FUNCTION_BLOCK _UDINT_TestSuite EXTENDS TcUnit.FB_TestSuite
VAR
END_VAR

TestAddress();
TestClearReference();
TestClone();
TestTypeNameReturnsExpected();
TestIsFloat();
TestIsSigned();
TestMakeReferenceToFollowsReference();
TestMakeReferenceToUpdatesReference();
TestSize();
TestValueReturnsExpectedAfterInit();
TestValueReturnsExpectedAfterChange();
TestSerializeTypeWith();
TestSerializeWith();
TestTryDeserializeFrom();
TestTryMakeReferenceToFollowsReference();
TestTryMakeReferenceToUpdatesReference();

METHOD PUBLIC TestAddress
VAR
    _type : _UDINT(0);
    notExpected : PVOID := 0;
    actual : PVOID;
END_VAR
TEST('TestAddress');

actual := _type.Address;

AssertFalse(
    Condition := (notExpected = actual),
    Message := 'Type did not return a valid address.'
);

TEST_FINISHED();
END_METHOD

METHOD PUBLIC TestClearReference
VAR
    _type : _UDINT(0);
	target : UDINT := 0;
    expected : UDINT := 0;
    actual : UDINT;
END_VAR
TEST('TestClearReference');

_type.MakeReferenceTo(target);
_type.ClearReference();
target := 123;

actual := _type.Value;

AssertEquals(
    Expected := expected,
    Actual := actual,
    Message := 'Value incorrectly followed target change'
);

TEST_FINISHED();
END_METHOD

METHOD PUBLIC TestClone
VAR
    _type : _UDINT(123);
	clone : I_Datatype;
	isValidClone : BOOL;
	compareResult : DINT;
END_VAR
TEST('TestClone');

clone := _type.Clone();

isValidClone := clone <> 0;

IF isValidClone THEN
	compareResult := memcmp(_type.Address, clone.Address, clone.Size);
END_IF

AssertTrue(
	Condition := isValidClone,
	Message := 'Clone did not produce a clone'
);

AssertEquals_DINT(
	Expected := 0,
    Actual := compareResult,
    Message := 'Clone did not return a valid clone.'
);

clone.Dispose();

TEST_FINISHED();
END_METHOD

METHOD PUBLIC TestIsFloat
VAR
    _type : _UDINT(0);
END_VAR
TEST('TestIsFloat');

AssertFalse(
	Condition := _type.IsFloat,
    Message := 'Type did not correctly identify itself as being unsigned'
);

TEST_FINISHED();
END_METHOD

METHOD PUBLIC TestIsSigned
VAR
    _type : _UDINT(0);
END_VAR
TEST('TestIsSigned');

AssertFalse(
	Condition := _type.IsSigned,
    Message := 'Type did not correctly identify itself as being unsigned'
);

TEST_FINISHED();
END_METHOD

METHOD PUBLIC TestMakeReferenceToFollowsReference
VAR
    _type : _UDINT(0);
	target : UDINT := 0;
    expected : UDINT := 123;
    actual : UDINT;
END_VAR
TEST('TestMakeReferenceToFollowsReference');

_type.MakeReferenceTo(target);
target := 123;

actual := _type.Value;

AssertEquals(
    Expected := expected,
    Actual := actual,
    Message := 'Value did not follow target change'
);

TEST_FINISHED();
END_METHOD

METHOD PUBLIC TestMakeReferenceToUpdatesReference
VAR
    _type : _UDINT(0);
	target : UDINT := 0;
    expected : UDINT := 123;
    actual : UDINT;
END_VAR
TEST('TestMakeReferenceToUpdatesReference');

_type.MakeReferenceTo(target);
_type.Value := 123;

actual := target;

AssertEquals(
    Expected := expected,
    Actual := actual,
    Message := 'Value did not update target'
);

TEST_FINISHED();
END_METHOD

METHOD PUBLIC TestSerializeTypeWith
VAR
    _type : _UDINT(0);
    serializer : JsonSerializer;
    expected : STRING(500) := '{"typeName":"UDINT","minValue":0,"maxValue":4294967295,"isSigned":false,"isFloat":false}';
    actual : STRING(500);
END_VAR
TEST('TestSerializeTypeWith');

serializer.Reset();
_type.SerializeTypeWith(serializer);
serializer.TryGetSerializedData(ADR(actual), SIZEOF(actual));

AssertEquals_STRING(
    Expected := expected,
    Actual := actual,
    Message := 'Serialization of type did not return correct string.'
);

TEST_FINISHED();
END_METHOD

METHOD PUBLIC TestSerializeWith
VAR
    _type : _UDINT(123);
    serializer : JsonSerializer;
    expected : STRING := '123';
    actual : STRING(500);
END_VAR
TEST('TestSerializeWith');

serializer.Reset();
_type.SerializeWith(serializer);
serializer.TryGetSerializedData(ADR(actual), SIZEOF(actual));

AssertEquals_STRING(
    Expected := expected,
    Actual := actual,
    Message := 'Serialization of type data did not return correct string.'
);

TEST_FINISHED();
END_METHOD

METHOD PUBLIC TestSize
VAR
    _type : _UDINT(0);
    expected : UDINT := SIZEOF(UDINT);
    actual : UDINT;
END_VAR
TEST('TestSize');

actual := _type.Size;

AssertEquals_UDINT(
    Expected := Expected,
    Actual := actual,
    Message := 'Type did not return the correct size.'
);

TEST_FINISHED();
END_METHOD

METHOD PUBLIC TestTryDeserializeFrom
VAR
    deserializer : JsonDeserializer;
    feedback : DeserializerFeedback;
    json : STRING := '123';
    _type : _UDINT(0);
    expected : UDINT := 123;
    actual : UDINT;
 END_VAR
TEST('TestTryDeserializeFrom');

deserializer.Reset();
deserializer.TryLoad(json);
_type.TryDeserializeFrom(Deserializer, Feedback);

actual := _type.Value;

AssertEquals(
    Expected := expected,
    Actual := actual,
    Message := 'Type did not deserialize correctly.'
);

TEST_FINISHED();
END_METHOD

METHOD PUBLIC TestTryMakeReferenceToFollowsReference
VAR
    _type : _UDINT(0);
	target : _UDINT(0);
    expected : UDINT := 123;
    actual : UDINT;
END_VAR
TEST('TestTryMakeReferenceToFollowsReference');

_type.TryMakeReferenceTo(target);
target.Value := 123;

actual := _type.Value;

AssertEquals(
    Expected := expected,
    Actual := actual,
    Message := 'Value did not follow target change'
);

TEST_FINISHED();
END_METHOD

METHOD PUBLIC TestTryMakeReferenceToUpdatesReference
VAR
    _type : _UDINT(0);
	target : _UDINT(0);
    expected : UDINT := 123;
    actual : UDINT;
END_VAR
TEST('TestTryMakeReferenceToUpdatesReference');

_type.TryMakeReferenceTo(target);
_type.Value := 123;

actual := target.Value;

AssertEquals(
    Expected := expected,
    Actual := actual,
    Message := 'Value did not update target'
);

TEST_FINISHED();
END_METHOD

METHOD PUBLIC TestTypeNameReturnsExpected
VAR
    _type : _UDINT(0);
    expected : STRING := 'UDINT';
    actual : STRING;
END_VAR
TEST('TestTypeNameReturnsExpected');

actual := _type.TypeName;

AssertEquals_STRING(
    Expected := expected,
    Actual := actual,
    Message := 'Type did not return correct iec type.'
);

TEST_FINISHED();
END_METHOD

METHOD PUBLIC TestValueReturnsExpectedAfterChange
VAR
    _type : _UDINT(0);
    expected : UDINT := 123;
    actual : UDINT;
END_VAR
TEST('TestValueReturnsExpectedAfterChange');

_type.Value := 123;

actual := _type.Value;

AssertEquals(
    Expected := expected,
    Actual := actual,
    Message := 'Expected value not returned after change.'
);

TEST_FINISHED();
END_METHOD

METHOD PUBLIC TestValueReturnsExpectedAfterInit
VAR
    _type : _UDINT(123);
    expected : UDINT := 123;
    actual : UDINT;
END_VAR
TEST('TestValueReturnsExpectedAfterInit');

actual := _type.Value;

AssertEquals(
    Expected := expected,
    Actual := actual,
    Message := 'Expected value not returned after Init.'
);

TEST_FINISHED();
END_METHOD

END_FUNCTION_BLOCK

(* stored: Version 1.1.0.1, ProductVersion 3.1.4024.12
   POU _UDINT_TestSuite: Id {2800a6ae-27d3-03ba-3911-8603c59c029a}, SpecialFunc None
   Method TestAddress: Id {99a2019e-ed45-0102-2932-822e518121fe}
   Method TestClearReference: Id {38937dd6-21b3-0552-20da-5c3d3787943e}
   Method TestClone: Id {b4d84e3b-1860-0841-3c59-7c02cd3bd047}
   Method TestIsFloat: Id {6e2992b0-27c6-462d-9092-3abdf0b287bb}
   Method TestIsSigned: Id {a661132e-a505-0f18-0177-1db667ec6b01}
   Method TestMakeReferenceToFollowsReference: Id {47c3d9a3-4886-0583-38d8-1ff279e5076a}
   Method TestMakeReferenceToUpdatesReference: Id {b107d813-75e4-0da0-3145-3fccfd7d3a1b}
   Method TestSerializeTypeWith: Id {82364cbe-7c0f-01f6-0916-3ed857cba279}
   Method TestSerializeWith: Id {34373aeb-43d7-0e1a-306d-5e5c4480e5f4}
   Method TestSize: Id {e70bf072-a655-0ac4-0f76-8affaf9cff94}
   Method TestTryDeserializeFrom: Id {486155b6-ff1b-013a-124e-88f87076fe7f}
   Method TestTryMakeReferenceToFollowsReference: Id {c482576f-2fdf-0690-3a5b-697c8e6c2029}
   Method TestTryMakeReferenceToUpdatesReference: Id {a75f484a-b38f-05cc-2ca8-14b1affbed78}
   Method TestTypeNameReturnsExpected: Id {605d4ae4-8bd5-02c8-376d-89e548e028a0}
   Method TestValueReturnsExpectedAfterChange: Id {d6b7b869-efc0-03f8-175c-3e4e28d2314b}
   Method TestValueReturnsExpectedAfterInit: Id {0cfe6839-4232-0c3a-2092-e63e0d7561fe} *)
